{region '#Template'}
	{attribute 'Version' := '1.0.0.0'}
	{attribute 'Tags' := '"LCID": "1031", "Text": "DUT, Room automation, Heating system"'}
	{attribute 'Tags' := '"LCID": "1033", "Text": "DUT, Room automation, Heating system"'}
	{attribute 'Description' := '"LCID": "1031", "Text": "Betriebsart Energieniveau"'}
	{attribute 'Description' := '"LCID": "1033", "Text": "Operating mode Energy level"'}
{endregion}

{attribute qualified_only}
TYPE E_BA_EnergyLvlEx :
(
	eProtection			:= 1,
	eEconomy			:= 2,
	ePreComfort			:= 3,
	eComfort			:= 4
	
) UDINT;
END_TYPE

(* stored: Version 1.1.0.1, ProductVersion 3.1.4024.9
   DUT E_BA_EnergyLvlEx: Id {b6f2cacb-c294-4ed1-8364-b983db3d500c} *)
